TYPE ST_ParamActionneur :
STRUCT
	tTimeOut : TIME; 			//max time allowed for moving to position bevor xState=TRUE
	xPresenceSensOut : BOOL; 	//If at the out-pos a Sensor is available
	xPresenceSensIn : BOOL; 	//If at the in-pos a Sensor is availaible
	tMoveOutTimeDelay : TIME; 	//delay after activating xPresenceSensOut before turning off output. When there is no Sensor, only this time will be used.
	tMoveInTimeDelay : TIME; 	//delay after activating xPresenceSensIn before turning off output. When there is no Sensor, only this time will be used.
END_STRUCT
END_TYPE

(* stored: Version 1.1.0.1, ProductVersion 3.1.4020.6
   DUT ST_ParamActionneur: Id {317ba1d7-24c1-4d0a-bd7c-4a300e6ce075} *)
